INTERFACE I_PtInterval

METHOD inMonth : DINT
VAR_INPUT
END_VAR
END_METHOD

METHOD inYears : DINT
VAR_INPUT
END_VAR
END_METHOD

END_INTERFACE

(* stored: Version 1.1.0.1, ProductVersion 3.1.4024.12
   Itf I_PtInterval: Id {05df78e9-3caa-4ed4-b96a-c677c020a88f}
   Method inMonth: Id {19cb2600-eff7-4586-a9f4-8c4d730cd521}
   Method inYears: Id {f5aeab6d-bcd1-4d1b-bf48-8f41929cc9bc} *)
